(* IEC 61131-3 sources: programs/VI-54/VI-54_20171205/VI-54_20171205/Stations/PLC_VI54/VI-54_171014/Class/RecipeBase, 1 file *)

(* ---- RecipeBase.st ---- *)
(*!
<Class
	Name               = "RecipeBase"
	Revision           = "0.0"
	RealtimeTask       = "false"
	CyclicTask         = "false"
	BackgroundTask     = "false"
	Sigmatek           = "false"
	OSInterface        = "false"
	HighPriority       = "false"
	Automatic          = "false"
	UpdateMode         = "Prescan"
	SharedCommandTable = "true"
	Objectsize         = "(284,120)">
	<Channels>
		<Server Name="Comm" Visualized="false" Initialize="false" WriteProtected="true" Retentive="false"/>
		<Client Name="MainRecipe" Required="true" Internal="false"/>
	</Channels>
</Class>
*)
RecipeBase : CLASS
  //Servers:
	Comm 	: SvrChCmd_DINT;
  //Clients:
	MainRecipe 	: CltChCmd_MainRecipe;
  //Variables:
		ReceptPtr 	: ^DataRecipeStr;
  //Functions:

	FUNCTION VIRTUAL GLOBAL Init;
  //Tables:
	FUNCTION @STD
		VAR_OUTPUT
			ret_code	: CONFSTATES;
		END_VAR;
	FUNCTION GLOBAL TAB @CT_;
END_CLASS;

#pragma usingLtd MainRecipe

FUNCTION VIRTUAL GLOBAL RecipeBase::Init

  if _FirstScan then
    ReceptPtr := MainRecipe.GetPointer();
  end_if;

END_FUNCTION
